PROGRAM HEATING
VAR
	HEATING1:FB_HEATING;
END_VAR


// GVL output koppelen
GVL.ox_HEATER :=HEATING1.HEATING;

HEATING1(ix_START:=GVL.ix_START,TEMP:=GVL.id_TEMP_SENSOR,
SETPOINT:=GVL.id_TEMP_SETPOINT);

END_PROGRAM

(* stored: Version 1.1.0.1, ProductVersion 3.1.4024.15
   POU HEATING: Id {8ac95230-94a2-43ca-860b-e38e82f2822b}, SpecialFunc None *)
